FUNCTION_BLOCK FB_UMWELT
VAR_INPUT
END_VAR
VAR_OUTPUT
END_VAR
VAR

	(*TF_aussen				: FB_TF;*)

	{attribute 'OPC.UA.DA' := '1'}Daemmerung				: REAL;
	{attribute 'OPC.UA.DA' := '1'}Temp_Aussen_WS_Mittelw	: REAL;
	{attribute 'OPC.UA.DA' := '1'}Temp_Aussen_WS			: REAL;
	{attribute 'OPC.UA.DA' := '1'}Regen					: BOOL;		
	{attribute 'OPC.UA.DA' := '1'}Windgeschwindigkeit		: REAL;

	(* Mittelwert	berechnung	: FB_CTRL_MOVING_AVERAGE;	*)

	{attribute 'OPC.UA.DA' := '1'}Temp_Aussen			: REAL;		
	{attribute 'OPC.UA.DA' := '1'}Temp_Aussen_Mittelw	: REAL;		
	{attribute 'OPC.UA.DA' := '1'}Temp_Halle_Sektor1		: REAL;	
	{attribute 'OPC.UA.DA' := '1'}Temp_Halle_Sektor2		: REAL;	
	{attribute 'OPC.UA.DA' := '1'}Temp_Halle_Sektor3		: REAL;	

	Tempfuehler_Halle_Sektor1				: FB_TF;
	Tempfuehler_Halle_Sektor2				: FB_TF;
	Tempfuehler_Halle_Sektor3				: FB_TF;
	Tempfuehler_Temperatur_Aussen_TF		: FB_TF;

	Tagesmittelung							: FB_UW_Temp_Mittelung;

END_VAR

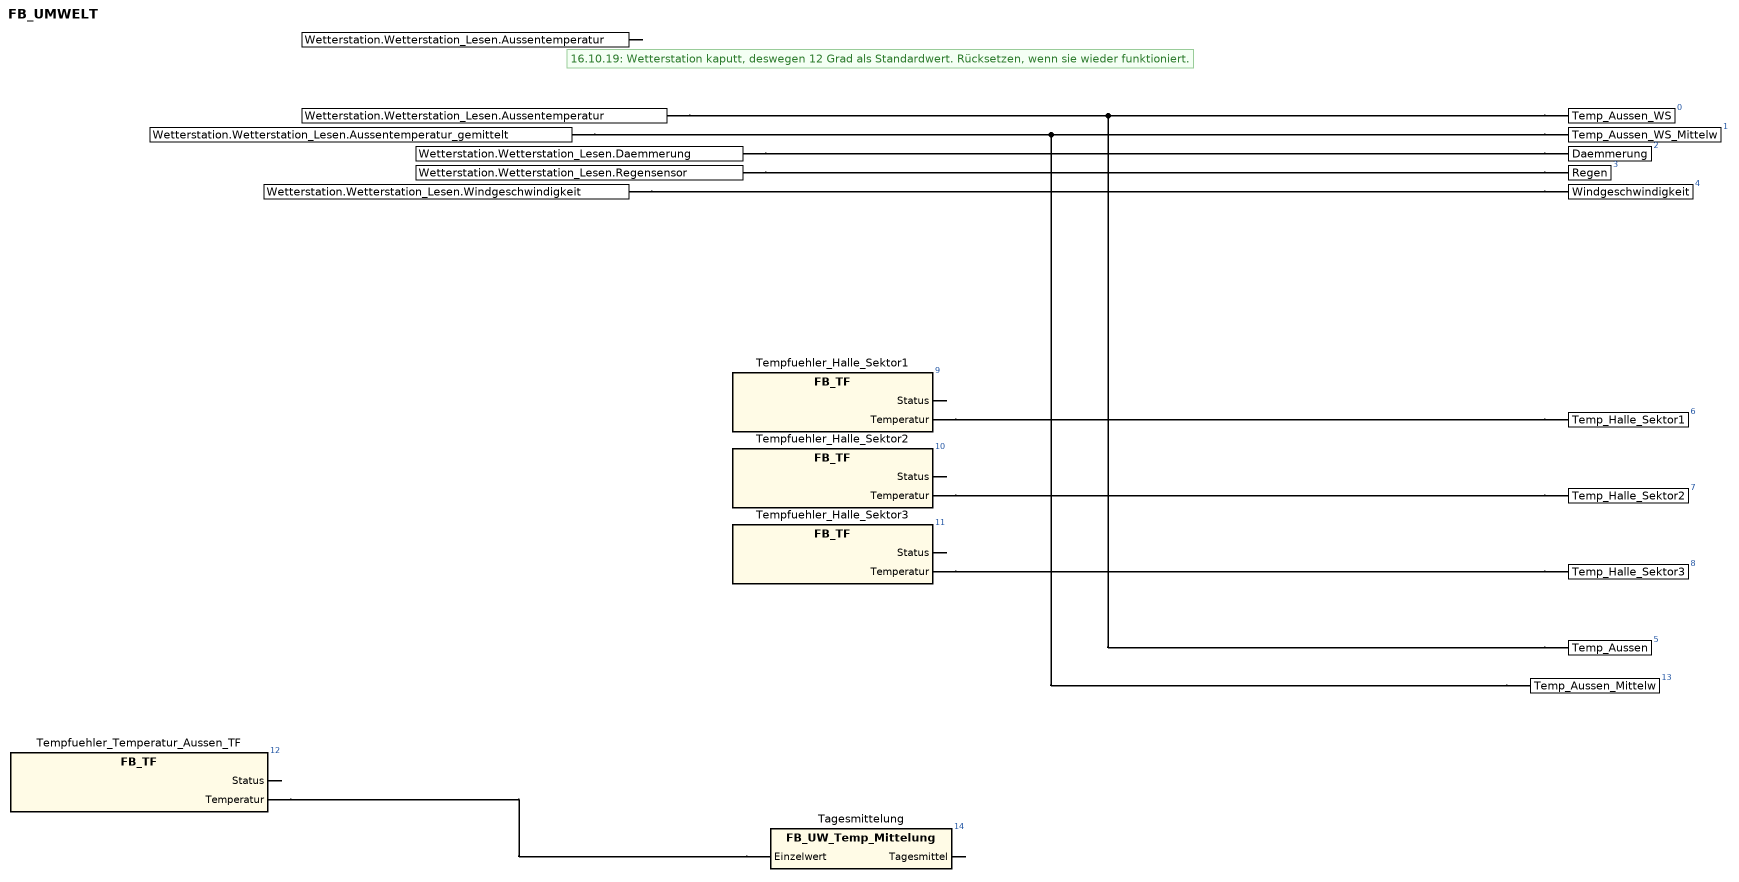
Temp_Aussen_WS := Wetterstation.Wetterstation_Lesen.Aussentemperatur;
Temp_Aussen_WS_Mittelw := Wetterstation.Wetterstation_Lesen.Aussentemperatur_gemittelt;
Daemmerung := Wetterstation.Wetterstation_Lesen.Daemmerung;
Regen := Wetterstation.Wetterstation_Lesen.Regensensor;
Windgeschwindigkeit := Wetterstation.Wetterstation_Lesen.Windgeschwindigkeit;
Temp_Aussen := Wetterstation.Wetterstation_Lesen.Aussentemperatur;
Temp_Halle_Sektor1 := Tempfuehler_Halle_Sektor1.Temperatur;
Temp_Halle_Sektor2 := Tempfuehler_Halle_Sektor2.Temperatur;
Temp_Halle_Sektor3 := Tempfuehler_Halle_Sektor3.Temperatur;
// 16.10.19: Wetterstation kaputt, deswegen 12 Grad als Standardwert. Rücksetzen, wenn sie wieder funktioniert.
Tempfuehler_Halle_Sektor1(); // FB_TF
Tempfuehler_Halle_Sektor2(); // FB_TF
Tempfuehler_Halle_Sektor3(); // FB_TF
Tempfuehler_Temperatur_Aussen_TF(); // FB_TF
Temp_Aussen_Mittelw := Wetterstation.Wetterstation_Lesen.Aussentemperatur_gemittelt;
Tagesmittelung(Einzelwert := Tempfuehler_Temperatur_Aussen_TF.Temperatur); // FB_UW_Temp_Mittelung
// Wetterstation.Wetterstation_Lesen.Aussentemperatur: input not connected

END_FUNCTION_BLOCK

(* stored: Version 1.1.0.1, ProductVersion 3.1.4024.9
   POU FB_UMWELT: Id {7b89a500-9296-4f75-a608-00a6b48a1294}, SpecialFunc None *)
